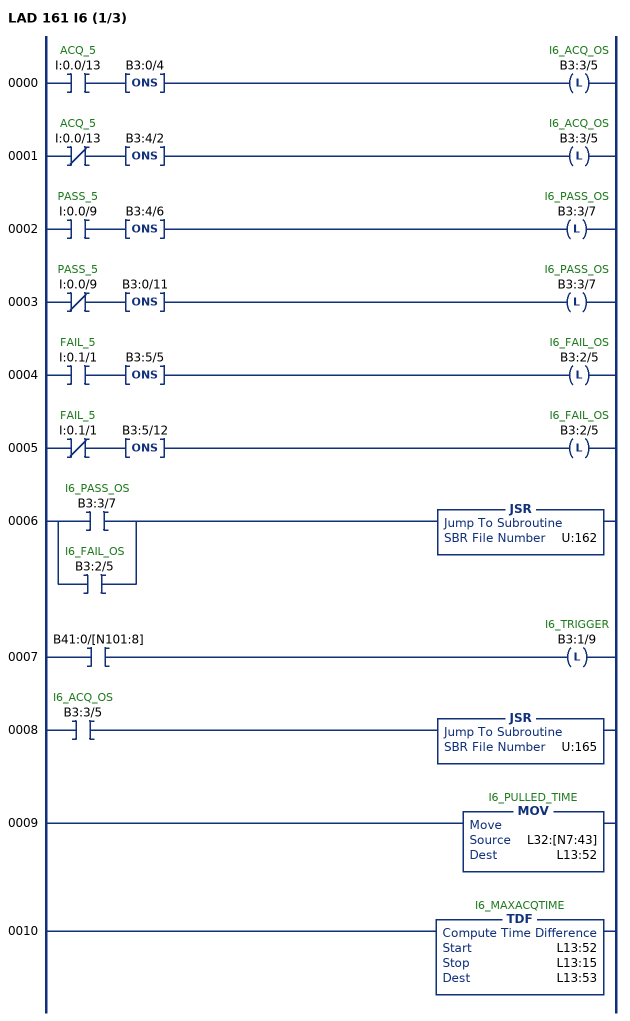
% Rung: 0 %
SOR XIC I:0.0/13 ONS B3:0/4 OTL B3:3/5 EOR
%   I:0.0/13  ACQ_5 %
%   B3:3/5  I6_ACQ_OS %
% Rung: 1 %
SOR XIO I:0.0/13 ONS B3:4/2 OTL B3:3/5 EOR
%   I:0.0/13  ACQ_5 %
%   B3:3/5  I6_ACQ_OS %
% Rung: 2 %
SOR XIC I:0.0/9 ONS B3:4/6 OTL B3:3/7 EOR
%   I:0.0/9  PASS_5 %
%   B3:3/7  I6_PASS_OS %
% Rung: 3 %
SOR XIO I:0.0/9 ONS B3:0/11 OTL B3:3/7 EOR
%   I:0.0/9  PASS_5 %
%   B3:3/7  I6_PASS_OS %
% Rung: 4 %
SOR XIC I:0.1/1 ONS B3:5/5 OTL B3:2/5 EOR
%   I:0.1/1  FAIL_5 %
%   B3:2/5  I6_FAIL_OS %
% Rung: 5 %
SOR XIO I:0.1/1 ONS B3:5/12 OTL B3:2/5 EOR
%   I:0.1/1  FAIL_5 %
%   B3:2/5  I6_FAIL_OS %
% Rung: 6 %
SOR BST XIC B3:3/7 NXB XIC B3:2/5 BND JSR U:162 EOR
%   B3:3/7  I6_PASS_OS %
%   B3:2/5  I6_FAIL_OS %
% Rung: 7 %
SOR XIC B41:0/[N101:8] OTL B3:1/9 EOR
%   B41:0  TOP_OK_3 %
%   N101:8  I6_TRIG_LOC %
%   B3:1/9  I6_TRIGGER %
% Rung: 8 %
SOR XIC B3:3/5 JSR U:165 EOR
%   B3:3/5  I6_ACQ_OS %
% Rung: 9 %
SOR MOV L32:[N7:43] L13:52 EOR
%   N7:43  I6_OLDEST_PART_INDEX %
%   L13:52  I6_PULLED_TIME %
% Rung: 10 %
SOR TDF L13:52 L13:15 L13:53 EOR
%   L13:52  I6_PULLED_TIME %
%   L13:15  THE_TIME %
%   L13:53  I6_MAXACQTIME %

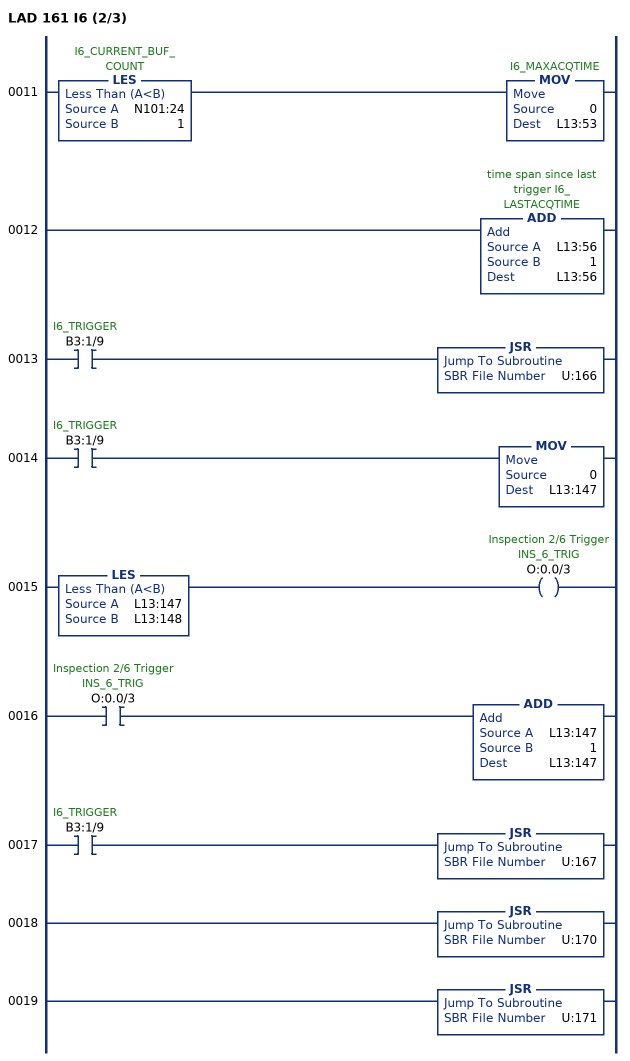
% Rung: 11 %
SOR LES N101:24 1 MOV 0 L13:53 EOR
%   N101:24  I6_CURRENT_BUF_COUNT %
%   L13:53  I6_MAXACQTIME %
% Rung: 12 %
SOR ADD L13:56 1 L13:56 EOR
%   L13:56  I6_LASTACQTIME  "time span since last trigger" %
% Rung: 13 %
SOR XIC B3:1/9 JSR U:166 EOR
%   B3:1/9  I6_TRIGGER %
% Rung: 14 %
SOR XIC B3:1/9 MOV 0 L13:147 EOR
%   B3:1/9  I6_TRIGGER %
% Rung: 15 %
SOR LES L13:147 L13:148 OTE O:0.0/3 EOR
%   O:0.0/3  INS_6_TRIG  "Inspection 2/6 Trigger" %
% Rung: 16 %
SOR XIC O:0.0/3 ADD L13:147 1 L13:147 EOR
%   O:0.0/3  INS_6_TRIG  "Inspection 2/6 Trigger" %
% Rung: 17 %
SOR XIC B3:1/9 JSR U:167 EOR
%   B3:1/9  I6_TRIGGER %
% Rung: 18 %
SOR JSR U:170 EOR
% Rung: 19 %
SOR JSR U:171 EOR

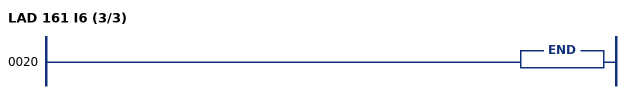
% Rung: 20 %
SOR END EOR

LADDER 162 "I6 RESULT"
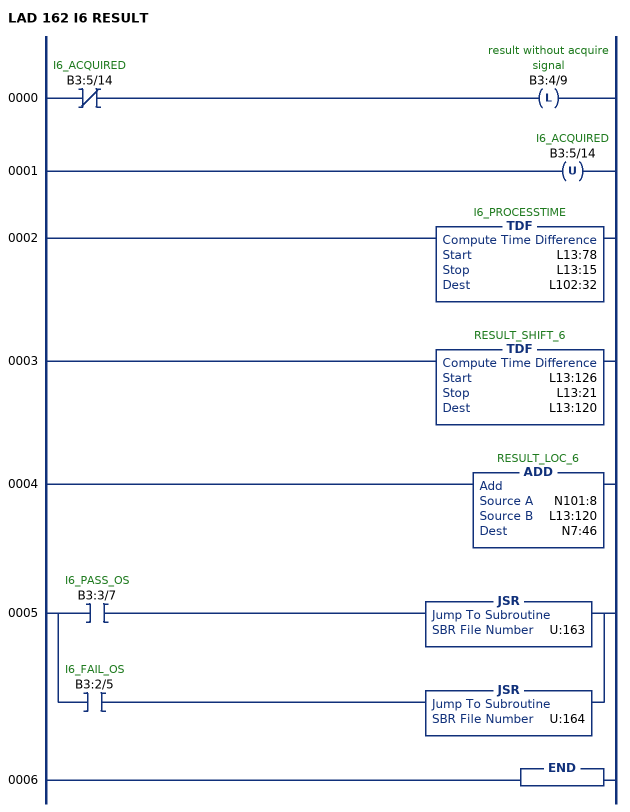
% Rung: 0 %
SOR XIO B3:5/14 OTL B3:4/9 EOR
%   B3:5/14  I6_ACQUIRED %
%   B3:4/9  "result without acquire signal" %
% Rung: 1 %
SOR OTU B3:5/14 EOR
%   B3:5/14  I6_ACQUIRED %
% Rung: 2 %
SOR TDF L13:78 L13:15 L102:32 EOR
%   L13:78  I6_TIMEOFACQ %
%   L13:15  THE_TIME %
%   L102:32  I6_PROCESSTIME %
% Rung: 3 %
SOR TDF L13:126 L13:21 L13:120 EOR
%   L13:126  I6_PROCESS_START_POS %
%   L13:21  TOP_POSITION %
%   L13:120  RESULT_SHIFT_6 %
% Rung: 4 %
SOR ADD N101:8 L13:120 N7:46 EOR
%   N101:8  I6_TRIG_LOC %
%   L13:120  RESULT_SHIFT_6 %
%   N7:46  RESULT_LOC_6 %
% Rung: 5 %
SOR BST XIC B3:3/7 JSR U:163 NXB XIC B3:2/5 JSR U:164 BND EOR
%   B3:3/7  I6_PASS_OS %
%   B3:2/5  I6_FAIL_OS %
% Rung: 6 %
SOR END EOR

LADDER 163 "I6 PASS"
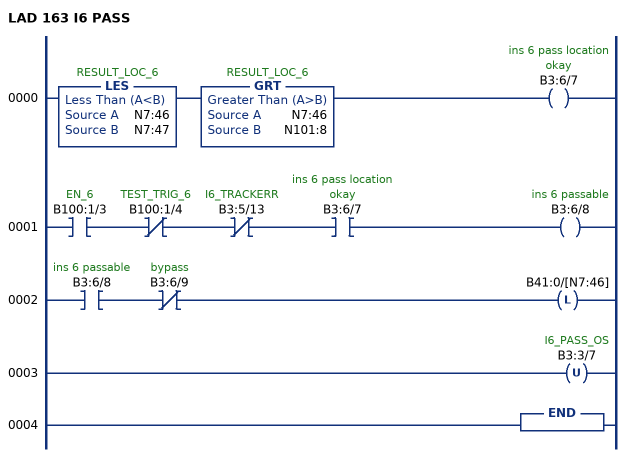
% Rung: 0 %
SOR LES N7:46 N7:47 GRT N7:46 N101:8 OTE B3:6/7 EOR
%   N7:46  RESULT_LOC_6 %
%   N7:47  I6_MAX_SHIFT  "ins 6 maximum result location" %
%   N101:8  I6_TRIG_LOC %
%   B3:6/7  "ins 6 pass location okay" %
% Rung: 1 %
SOR XIC B100:1/3 XIO B100:1/4 XIO B3:5/13 XIC B3:6/7 OTE B3:6/8 EOR
%   B100:1/3  EN_6 %
%   B100:1/4  TEST_TRIG_6 %
%   B3:5/13  I6_TRACKERR %
%   B3:6/7  "ins 6 pass location okay" %
%   B3:6/8  "ins 6 passable" %
% Rung: 2 %
SOR XIC B3:6/8 XIO B3:6/9 OTL B41:0/[N7:46] EOR
%   B3:6/8  "ins 6 passable" %
%   B3:6/9  "bypass" %
%   B41:0  TOP_OK_3 %
%   N7:46  RESULT_LOC_6 %
% Rung: 3 %
SOR OTU B3:3/7 EOR
%   B3:3/7  I6_PASS_OS %
% Rung: 4 %
SOR END EOR

LADDER 164 "I6 FAIL"
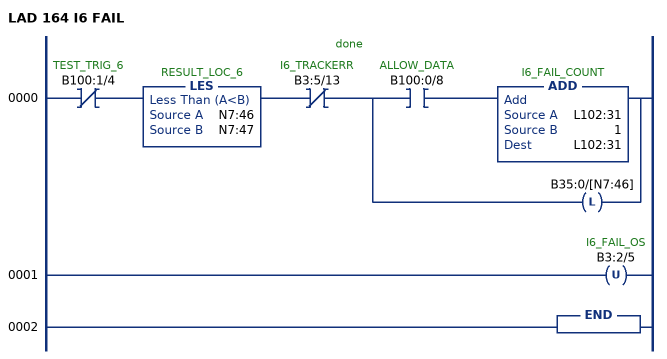
% Rung: 0 %
% done %
SOR XIO B100:1/4 LES N7:46 N7:47 XIO B3:5/13 BST XIC B100:0/8 ADD L102:31 1 L102:31 NXB OTL B35:0/[N7:46] BND EOR
%   B100:1/4  TEST_TRIG_6 %
%   N7:46  RESULT_LOC_6 %
%   N7:47  I6_MAX_SHIFT  "ins 6 maximum result location" %
%   B3:5/13  I6_TRACKERR %
%   B100:0/8  ALLOW_DATA %
%   L102:31  I6_FAIL_COUNT %
%   B35:0  TOP_NG %
% Rung: 1 %
SOR OTU B3:2/5 EOR
%   B3:2/5  I6_FAIL_OS %
% Rung: 2 %
SOR END EOR

LADDER 165 "I6 ACQ"
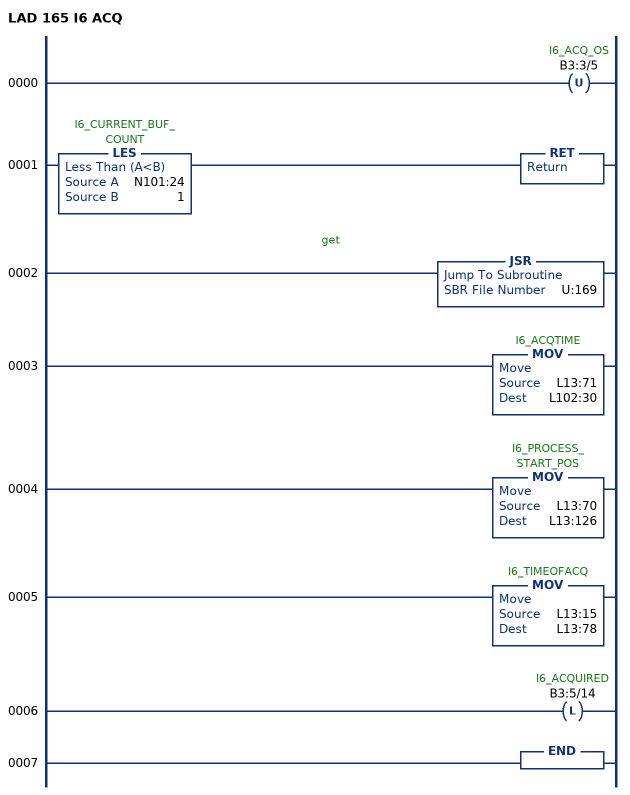
% Rung: 0 %
SOR OTU B3:3/5 EOR
%   B3:3/5  I6_ACQ_OS %
% Rung: 1 %
SOR LES N101:24 1 RET EOR
%   N101:24  I6_CURRENT_BUF_COUNT %
% Rung: 2 %
% get %
SOR JSR U:169 EOR
% Rung: 3 %
SOR MOV L13:71 L102:30 EOR
%   L13:71  I6_TIME_SPAN %
%   L102:30  I6_ACQTIME %
% Rung: 4 %
SOR MOV L13:70 L13:126 EOR
%   L13:70  I6_PULLED_POSITION %
%   L13:126  I6_PROCESS_START_POS %
% Rung: 5 %
SOR MOV L13:15 L13:78 EOR
%   L13:15  THE_TIME %
%   L13:78  I6_TIMEOFACQ %
% Rung: 6 %
SOR OTL B3:5/14 EOR
%   B3:5/14  I6_ACQUIRED %
% Rung: 7 %
SOR END EOR

LADDER 166 "I6 TESTER"
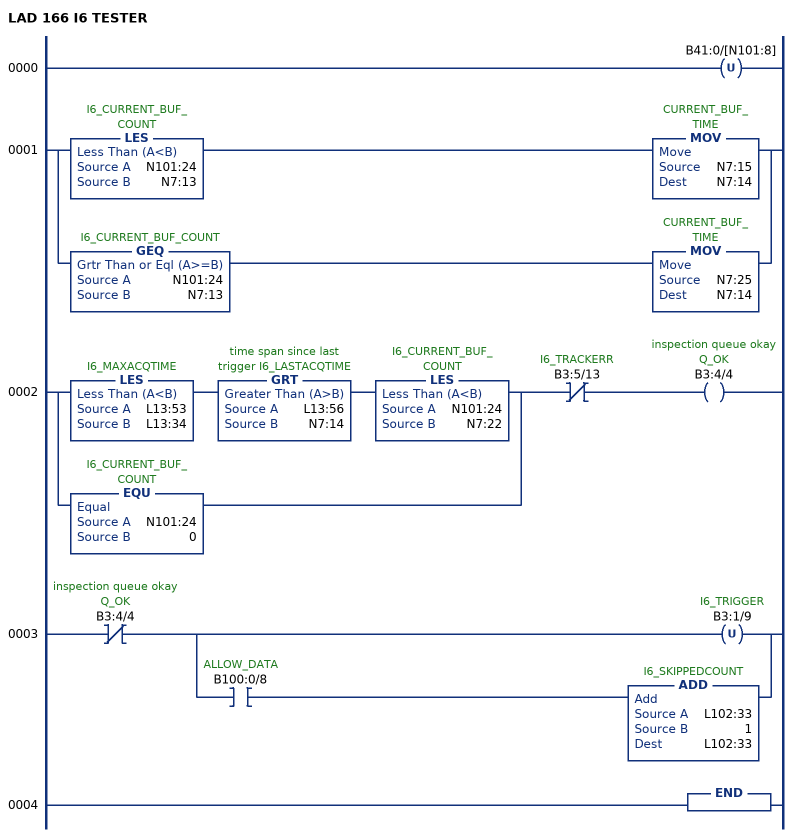
% Rung: 0 %
SOR OTU B41:0/[N101:8] EOR
%   B41:0  TOP_OK_3 %
%   N101:8  I6_TRIG_LOC %
% Rung: 1 %
SOR BST LES N101:24 N7:13 MOV N7:15 N7:14 NXB GEQ N101:24 N7:13 MOV N7:25 N7:14 BND EOR
%   N101:24  I6_CURRENT_BUF_COUNT %
%   N7:13  BUF_TRANS  "cam to pc buf transition" %
%   N7:15  CAM_BUF_TIME  "cam buf time" %
%   N7:14  CURRENT_BUF_TIME %
%   N7:25  PC_BUF_TIME  "pc buf time" %
% Rung: 2 %
SOR BST LES L13:53 L13:34 GRT L13:56 N7:14 LES N101:24 N7:22 NXB EQU N101:24 0 BND XIO B3:5/13 OTE B3:4/4 EOR
%   L13:53  I6_MAXACQTIME %
%   L13:34  MAX_ACQ_ALL  "absolute max acquire time before bypass trigger" %
%   L13:56  I6_LASTACQTIME  "time span since last trigger" %
%   N7:14  CURRENT_BUF_TIME %
%   N101:24  I6_CURRENT_BUF_COUNT %
%   N7:22  MAX_BUF_ALL  "max buffer count alowed before bypass" %
%   B3:5/13  I6_TRACKERR %
%   B3:4/4  Q_OK  "inspection queue okay" %
% Rung: 3 %
SOR XIO B3:4/4 BST OTU B3:1/9 NXB XIC B100:0/8 ADD L102:33 1 L102:33 BND EOR
%   B3:4/4  Q_OK  "inspection queue okay" %
%   B3:1/9  I6_TRIGGER %
%   B100:0/8  ALLOW_DATA %
%   L102:33  I6_SKIPPEDCOUNT %
% Rung: 4 %
SOR END EOR

LADDER 167 "I6 TRIG"
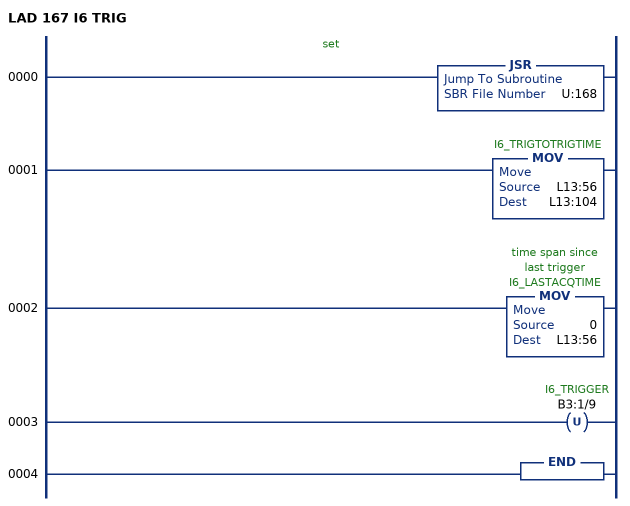
% Rung: 0 %
% set %
SOR JSR U:168 EOR
% Rung: 1 %
SOR MOV L13:56 L13:104 EOR
%   L13:56  I6_LASTACQTIME  "time span since last trigger" %
%   L13:104  I6_TRIGTOTRIGTIME %
% Rung: 2 %
SOR MOV 0 L13:56 EOR
%   L13:56  I6_LASTACQTIME  "time span since last trigger" %
% Rung: 3 %
SOR OTU B3:1/9 EOR
%   B3:1/9  I6_TRIGGER %
% Rung: 4 %
SOR END EOR

LADDER 168 "I6 FIFOSET"
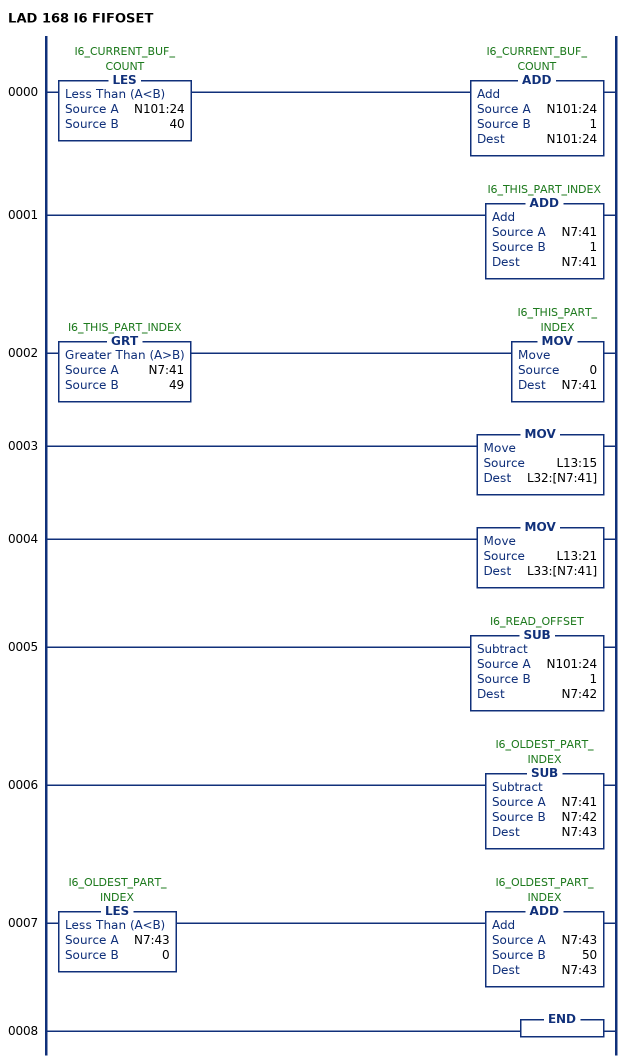
% Rung: 0 %
SOR LES N101:24 40 ADD N101:24 1 N101:24 EOR
%   N101:24  I6_CURRENT_BUF_COUNT %
% Rung: 1 %
SOR ADD N7:41 1 N7:41 EOR
%   N7:41  I6_THIS_PART_INDEX %
% Rung: 2 %
SOR GRT N7:41 49 MOV 0 N7:41 EOR
%   N7:41  I6_THIS_PART_INDEX %
% Rung: 3 %
SOR MOV L13:15 L32:[N7:41] EOR
%   L13:15  THE_TIME %
%   N7:41  I6_THIS_PART_INDEX %
% Rung: 4 %
SOR MOV L13:21 L33:[N7:41] EOR
%   L13:21  TOP_POSITION %
%   N7:41  I6_THIS_PART_INDEX %
% Rung: 5 %
SOR SUB N101:24 1 N7:42 EOR
%   N101:24  I6_CURRENT_BUF_COUNT %
%   N7:42  I6_READ_OFFSET %
% Rung: 6 %
SOR SUB N7:41 N7:42 N7:43 EOR
%   N7:41  I6_THIS_PART_INDEX %
%   N7:42  I6_READ_OFFSET %
%   N7:43  I6_OLDEST_PART_INDEX %
% Rung: 7 %
SOR LES N7:43 0 ADD N7:43 50 N7:43 EOR
%   N7:43  I6_OLDEST_PART_INDEX %
% Rung: 8 %
SOR END EOR

LADDER 169 "I6 FIFOGET"
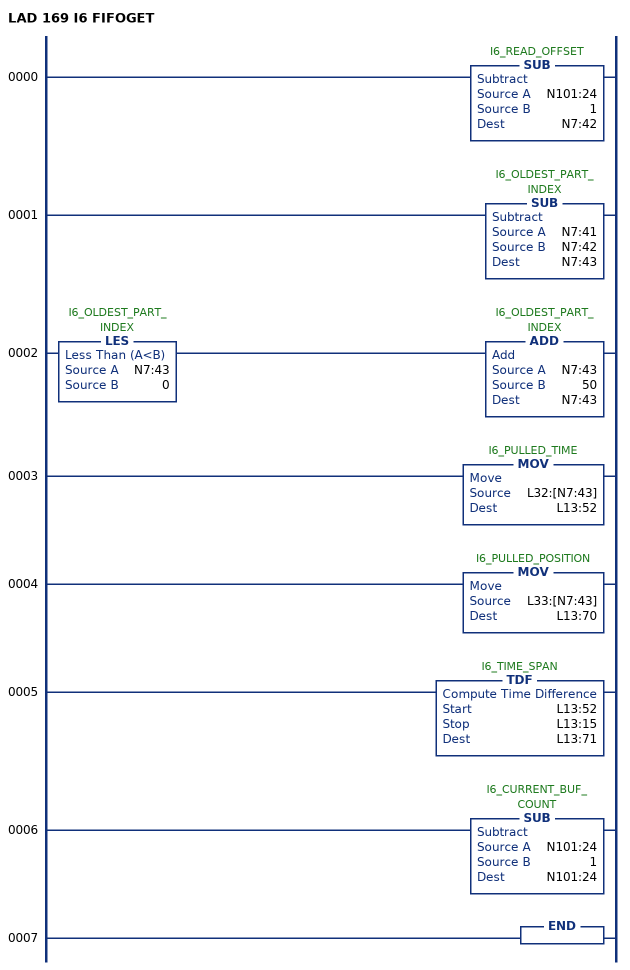
% Rung: 0 %
SOR SUB N101:24 1 N7:42 EOR
%   N101:24  I6_CURRENT_BUF_COUNT %
%   N7:42  I6_READ_OFFSET %
% Rung: 1 %
SOR SUB N7:41 N7:42 N7:43 EOR
%   N7:41  I6_THIS_PART_INDEX %
%   N7:42  I6_READ_OFFSET %
%   N7:43  I6_OLDEST_PART_INDEX %
% Rung: 2 %
SOR LES N7:43 0 ADD N7:43 50 N7:43 EOR
%   N7:43  I6_OLDEST_PART_INDEX %
% Rung: 3 %
SOR MOV L32:[N7:43] L13:52 EOR
%   N7:43  I6_OLDEST_PART_INDEX %
%   L13:52  I6_PULLED_TIME %
% Rung: 4 %
SOR MOV L33:[N7:43] L13:70 EOR
%   N7:43  I6_OLDEST_PART_INDEX %
%   L13:70  I6_PULLED_POSITION %
% Rung: 5 %
SOR TDF L13:52 L13:15 L13:71 EOR
%   L13:52  I6_PULLED_TIME %
%   L13:15  THE_TIME %
%   L13:71  I6_TIME_SPAN %
% Rung: 6 %
SOR SUB N101:24 1 N101:24 EOR
%   N101:24  I6_CURRENT_BUF_COUNT %
% Rung: 7 %
SOR END EOR

LADDER 170 "I6 DATA"
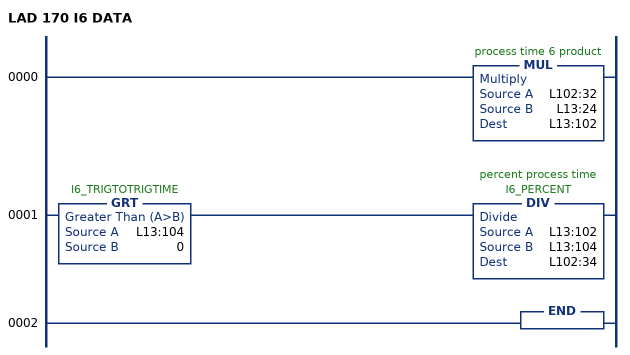
% Rung: 0 %
SOR MUL L102:32 L13:24 L13:102 EOR
%   L102:32  I6_PROCESSTIME %
%   L13:24  "multiplyer to make devision come out to a percentage" %
%   L13:102  "process time 6 product" %
% Rung: 1 %
SOR GRT L13:104 0 DIV L13:102 L13:104 L102:34 EOR
%   L13:104  I6_TRIGTOTRIGTIME %
%   L13:102  "process time 6 product" %
%   L102:34  I6_PERCENT  "percent process time" %
% Rung: 2 %
SOR END EOR

LADDER 171 "I6 FAULT"
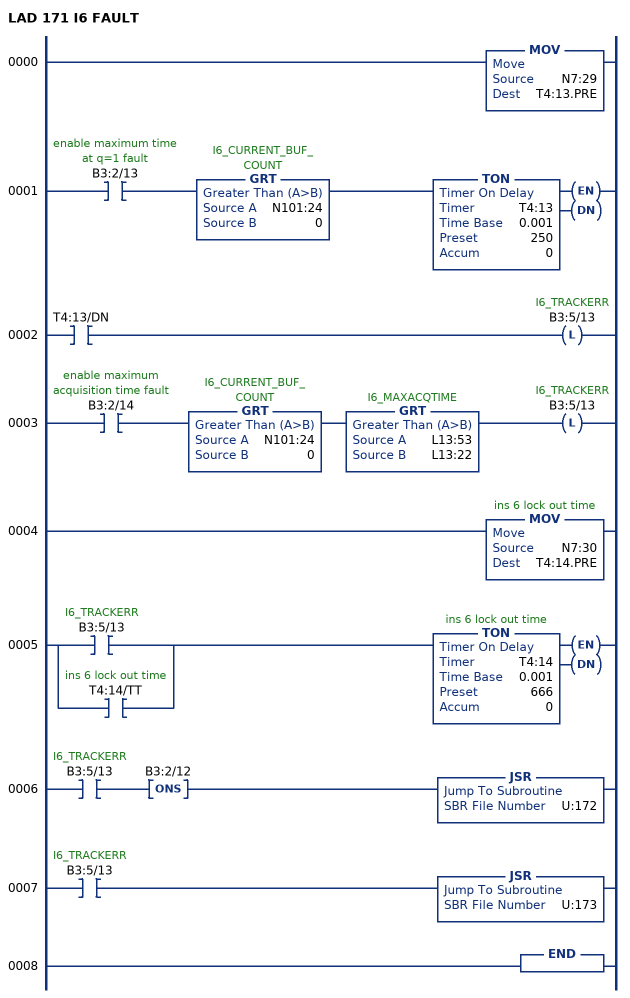
% Rung: 0 %
SOR MOV N7:29 T4:13.PRE EOR
%   N7:29  "max allowed ms time for q to be above 1 if safe fault is used" %
% Rung: 1 %
SOR XIC B3:2/13 GRT N101:24 0 TON T4:13 0.001 250 0 EOR
%   B3:2/13  "enable maximum time at q=1 fault" %
%   N101:24  I6_CURRENT_BUF_COUNT %
% Rung: 2 %
SOR XIC T4:13/DN OTL B3:5/13 EOR
%   B3:5/13  I6_TRACKERR %
% Rung: 3 %
SOR XIC B3:2/14 GRT N101:24 0 GRT L13:53 L13:22 OTL B3:5/13 EOR
%   B3:2/14  "enable maximum acquisition time fault" %
%   N101:24  I6_CURRENT_BUF_COUNT %
%   L13:53  I6_MAXACQTIME %
%   L13:22  "maximum of the longest acquire time allowed if maximum acquire time fault is enabled" %
%   B3:5/13  I6_TRACKERR %
% Rung: 4 %
SOR MOV N7:30 T4:14.PRE EOR
%   N7:30  "ms time setting to lock out inspection to give all pending images a chance to clear" %
%   T4:14  "ins 6 lock out time" %
% Rung: 5 %
SOR BST XIC B3:5/13 NXB XIC T4:14/TT BND TON T4:14 0.001 666 0 EOR
%   B3:5/13  I6_TRACKERR %
%   T4:14  "ins 6 lock out time" %
% Rung: 6 %
SOR XIC B3:5/13 ONS B3:2/12 JSR U:172 EOR
%   B3:5/13  I6_TRACKERR %
% Rung: 7 %
SOR XIC B3:5/13 JSR U:173 EOR
%   B3:5/13  I6_TRACKERR %
% Rung: 8 %
SOR END EOR

LADDER 172 "I6 FIX1"
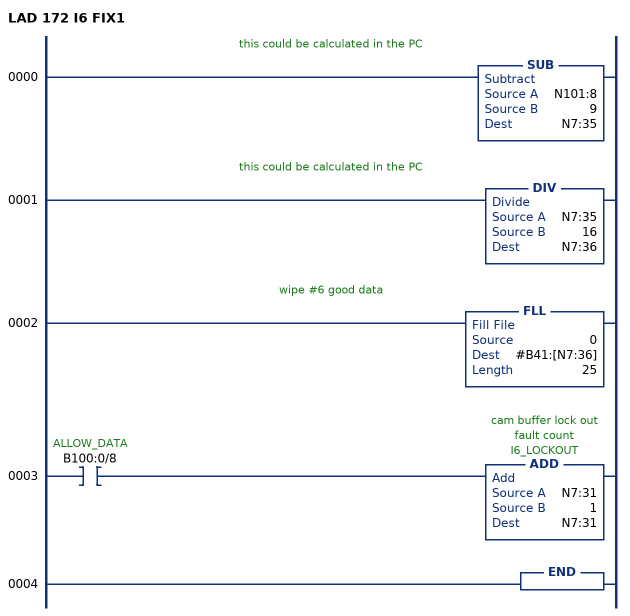
% Rung: 0 %
% this could be calculated in the PC %
SOR SUB N101:8 9 N7:35 EOR
%   N101:8  I6_TRIG_LOC %
% Rung: 1 %
% this could be calculated in the PC %
SOR DIV N7:35 16 N7:36 EOR
% Rung: 2 %
% wipe #6 good data %
SOR FLL 0 #B41:[N7:36] 25 EOR
% Rung: 3 %
SOR XIC B100:0/8 ADD N7:31 1 N7:31 EOR
%   B100:0/8  ALLOW_DATA %
%   N7:31  I6_LOCKOUT  "cam buffer lock out fault count" %
% Rung: 4 %
SOR END EOR

LADDER 173 "I6 FIX2"
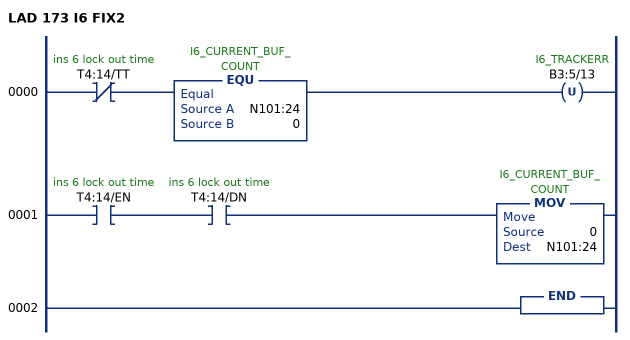
% Rung: 0 %
SOR XIO T4:14/TT EQU N101:24 0 OTU B3:5/13 EOR
%   T4:14  "ins 6 lock out time" %
%   N101:24  I6_CURRENT_BUF_COUNT %
%   B3:5/13  I6_TRACKERR %
% Rung: 1 %
SOR XIC T4:14/EN XIC T4:14/DN MOV 0 N101:24 EOR
%   T4:14  "ins 6 lock out time" %
%   N101:24  I6_CURRENT_BUF_COUNT %
% Rung: 2 %
SOR END EOR

LADDER 174 "I7"
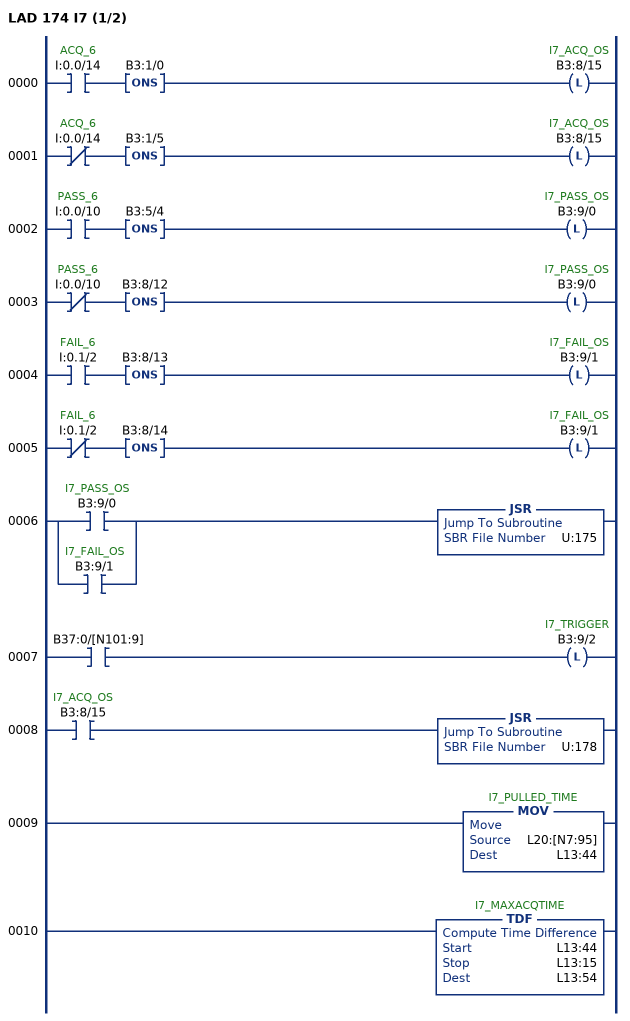
% Rung: 0 %
SOR XIC I:0.0/14 ONS B3:1/0 OTL B3:8/15 EOR
%   I:0.0/14  ACQ_6 %
%   B3:8/15  I7_ACQ_OS %
% Rung: 1 %
SOR XIO I:0.0/14 ONS B3:1/5 OTL B3:8/15 EOR
%   I:0.0/14  ACQ_6 %
%   B3:8/15  I7_ACQ_OS %
% Rung: 2 %
SOR XIC I:0.0/10 ONS B3:5/4 OTL B3:9/0 EOR
%   I:0.0/10  PASS_6 %
%   B3:9/0  I7_PASS_OS %
% Rung: 3 %
SOR XIO I:0.0/10 ONS B3:8/12 OTL B3:9/0 EOR
%   I:0.0/10  PASS_6 %
%   B3:9/0  I7_PASS_OS %
% Rung: 4 %
SOR XIC I:0.1/2 ONS B3:8/13 OTL B3:9/1 EOR
%   I:0.1/2  FAIL_6 %
%   B3:9/1  I7_FAIL_OS %
% Rung: 5 %
SOR XIO I:0.1/2 ONS B3:8/14 OTL B3:9/1 EOR
%   I:0.1/2  FAIL_6 %
%   B3:9/1  I7_FAIL_OS %
% Rung: 6 %
SOR BST XIC B3:9/0 NXB XIC B3:9/1 BND JSR U:175 EOR
%   B3:9/0  I7_PASS_OS %
%   B3:9/1  I7_FAIL_OS %
% Rung: 7 %
SOR XIC B37:0/[N101:9] OTL B3:9/2 EOR
%   B37:0  TOP_OK_1 %
%   N101:9  I7_TRIG_LOC %
%   B3:9/2  I7_TRIGGER %
% Rung: 8 %
SOR XIC B3:8/15 JSR U:178 EOR
%   B3:8/15  I7_ACQ_OS %
% Rung: 9 %
SOR MOV L20:[N7:95] L13:44 EOR
%   N7:95  I7_OLDEST_PART_INDEX %
%   L13:44  I7_PULLED_TIME %
% Rung: 10 %
SOR TDF L13:44 L13:15 L13:54 EOR
%   L13:44  I7_PULLED_TIME %
%   L13:15  THE_TIME %
%   L13:54  I7_MAXACQTIME %

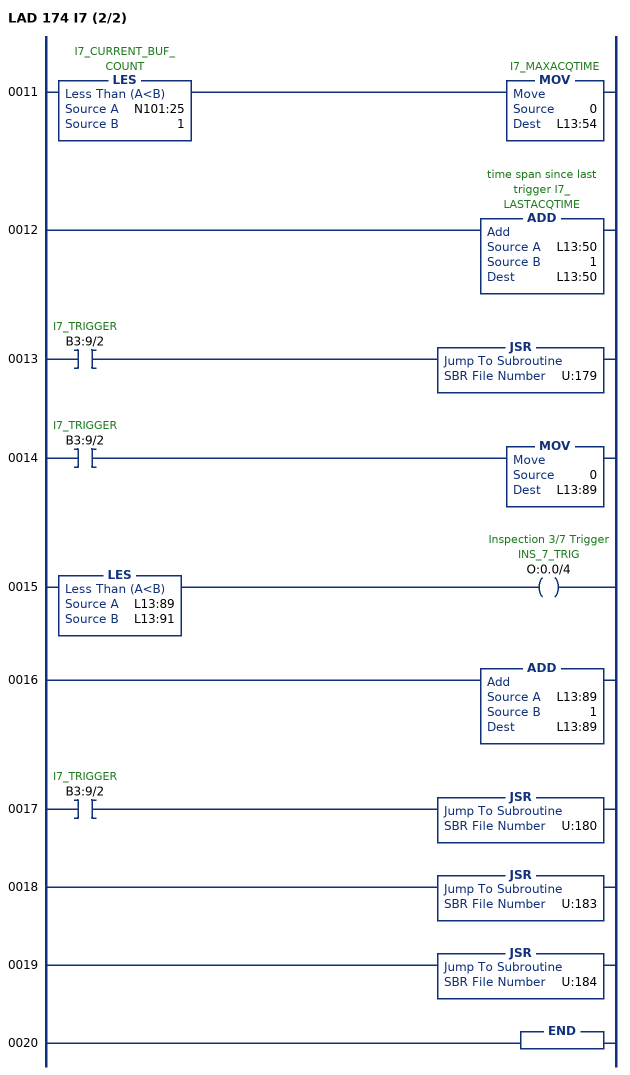
% Rung: 11 %
SOR LES N101:25 1 MOV 0 L13:54 EOR
%   N101:25  I7_CURRENT_BUF_COUNT %
%   L13:54  I7_MAXACQTIME %
% Rung: 12 %
SOR ADD L13:50 1 L13:50 EOR
%   L13:50  I7_LASTACQTIME  "time span since last trigger" %
% Rung: 13 %
SOR XIC B3:9/2 JSR U:179 EOR
%   B3:9/2  I7_TRIGGER %
% Rung: 14 %
SOR XIC B3:9/2 MOV 0 L13:89 EOR
%   B3:9/2  I7_TRIGGER %
% Rung: 15 %
SOR LES L13:89 L13:91 OTE O:0.0/4 EOR
%   L13:91  "test fire interval index" %
%   O:0.0/4  INS_7_TRIG  "Inspection 3/7 Trigger" %
% Rung: 16 %
SOR ADD L13:89 1 L13:89 EOR
% Rung: 17 %
SOR XIC B3:9/2 JSR U:180 EOR
%   B3:9/2  I7_TRIGGER %
% Rung: 18 %
SOR JSR U:183 EOR
% Rung: 19 %
SOR JSR U:184 EOR
% Rung: 20 %
SOR END EOR

LADDER 175 "I7 RESULT"
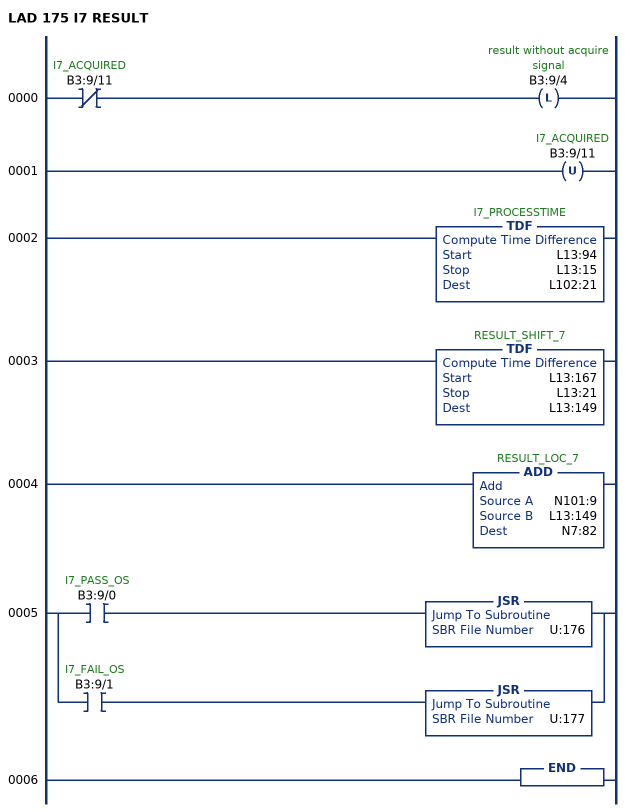
% Rung: 0 %
SOR XIO B3:9/11 OTL B3:9/4 EOR
%   B3:9/11  I7_ACQUIRED %
%   B3:9/4  "result without acquire signal" %
% Rung: 1 %
SOR OTU B3:9/11 EOR
%   B3:9/11  I7_ACQUIRED %
% Rung: 2 %
SOR TDF L13:94 L13:15 L102:21 EOR
%   L13:94  I7_TIMEOFACQ %
%   L13:15  THE_TIME %
%   L102:21  I7_PROCESSTIME %
% Rung: 3 %
SOR TDF L13:167 L13:21 L13:149 EOR
%   L13:167  I7_PROCESS_START_POS %
%   L13:21  TOP_POSITION %
%   L13:149  RESULT_SHIFT_7 %
% Rung: 4 %
SOR ADD N101:9 L13:149 N7:82 EOR
%   N101:9  I7_TRIG_LOC %
%   L13:149  RESULT_SHIFT_7 %
%   N7:82  RESULT_LOC_7 %
% Rung: 5 %
SOR BST XIC B3:9/0 JSR U:176 NXB XIC B3:9/1 JSR U:177 BND EOR
%   B3:9/0  I7_PASS_OS %
%   B3:9/1  I7_FAIL_OS %
% Rung: 6 %
SOR END EOR

LADDER 176 "I7 PASS"
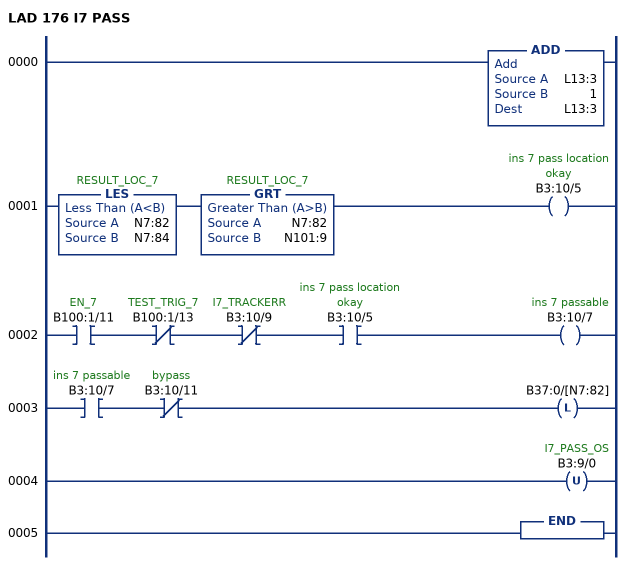
% Rung: 0 %
SOR ADD L13:3 1 L13:3 EOR
% Rung: 1 %
SOR LES N7:82 N7:84 GRT N7:82 N101:9 OTE B3:10/5 EOR
%   N7:82  RESULT_LOC_7 %
%   N7:84  I7_MAX_SHIFT %
%   N101:9  I7_TRIG_LOC %
%   B3:10/5  "ins 7 pass location okay" %
% Rung: 2 %
SOR XIC B100:1/11 XIO B100:1/13 XIO B3:10/9 XIC B3:10/5 OTE B3:10/7 EOR
%   B100:1/11  EN_7 %
%   B100:1/13  TEST_TRIG_7 %
%   B3:10/9  I7_TRACKERR %
%   B3:10/5  "ins 7 pass location okay" %
%   B3:10/7  "ins 7 passable" %
% Rung: 3 %
SOR XIC B3:10/7 XIO B3:10/11 OTL B37:0/[N7:82] EOR
%   B3:10/7  "ins 7 passable" %
%   B3:10/11  "bypass" %
%   B37:0  TOP_OK_1 %
%   N7:82  RESULT_LOC_7 %
% Rung: 4 %
SOR OTU B3:9/0 EOR
%   B3:9/0  I7_PASS_OS %
% Rung: 5 %
SOR END EOR

LADDER 177 "I7 FAIL"
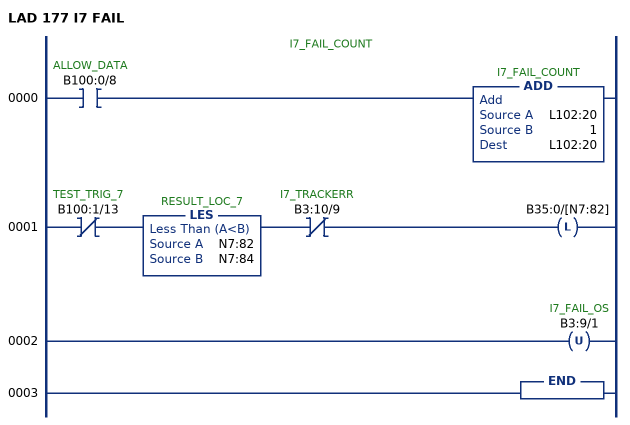
% Rung: 0 %
% I7_FAIL_COUNT %
SOR XIC B100:0/8 ADD L102:20 1 L102:20 EOR
%   B100:0/8  ALLOW_DATA %
%   L102:20  I7_FAIL_COUNT %
% Rung: 1 %
SOR XIO B100:1/13 LES N7:82 N7:84 XIO B3:10/9 OTL B35:0/[N7:82] EOR
%   B100:1/13  TEST_TRIG_7 %
%   N7:82  RESULT_LOC_7 %
%   N7:84  I7_MAX_SHIFT %
%   B3:10/9  I7_TRACKERR %
%   B35:0  TOP_NG %
% Rung: 2 %
SOR OTU B3:9/1 EOR
%   B3:9/1  I7_FAIL_OS %
% Rung: 3 %
SOR END EOR

LADDER 178 "I7 ACQ"
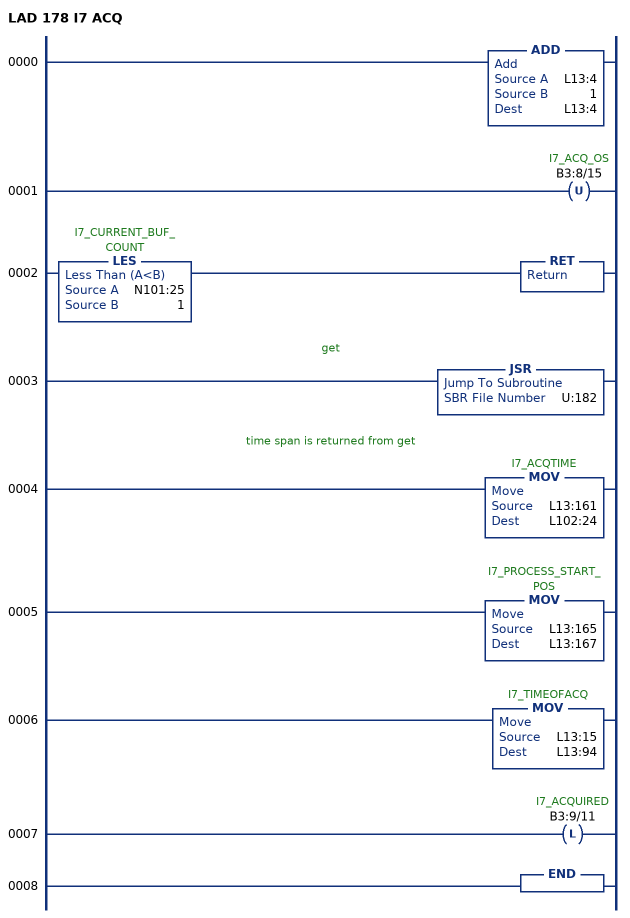
% Rung: 0 %
SOR ADD L13:4 1 L13:4 EOR
% Rung: 1 %
SOR OTU B3:8/15 EOR
%   B3:8/15  I7_ACQ_OS %
% Rung: 2 %
SOR LES N101:25 1 RET EOR
%   N101:25  I7_CURRENT_BUF_COUNT %
% Rung: 3 %
% get %
SOR JSR U:182 EOR
% Rung: 4 %
% time span is returned from get %
SOR MOV L13:161 L102:24 EOR
%   L13:161  I7_TIME_SPAN %
%   L102:24  I7_ACQTIME %
% Rung: 5 %
SOR MOV L13:165 L13:167 EOR
%   L13:165  I7_PULLED_POSITION %
%   L13:167  I7_PROCESS_START_POS %
% Rung: 6 %
SOR MOV L13:15 L13:94 EOR
%   L13:15  THE_TIME %
%   L13:94  I7_TIMEOFACQ %
% Rung: 7 %
SOR OTL B3:9/11 EOR
%   B3:9/11  I7_ACQUIRED %
% Rung: 8 %
SOR END EOR

LADDER 179 "I7 TESTER"
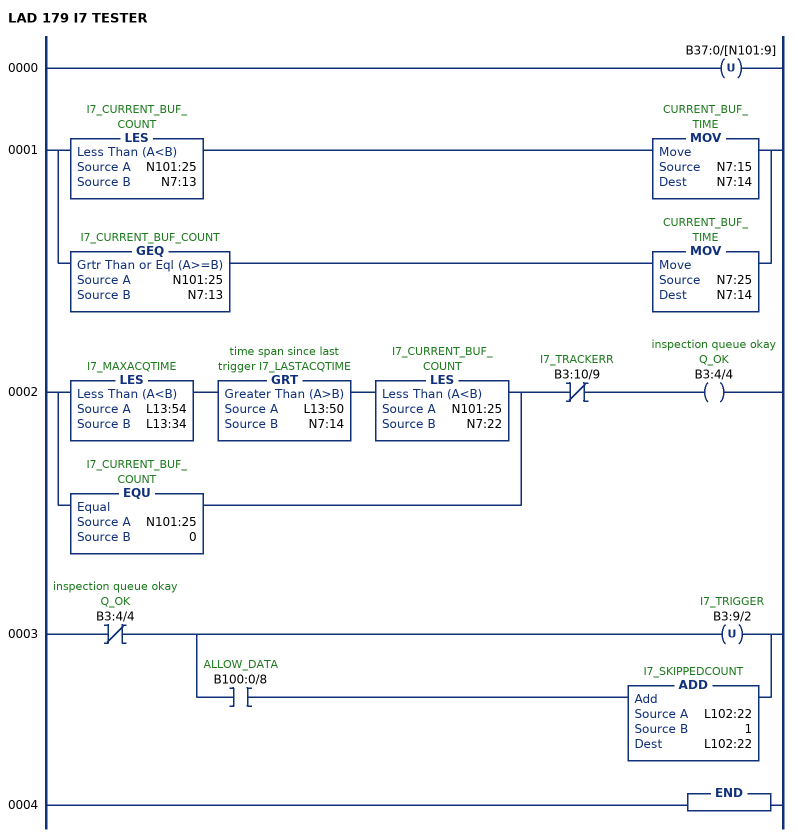
% Rung: 0 %
SOR OTU B37:0/[N101:9] EOR
%   B37:0  TOP_OK_1 %
%   N101:9  I7_TRIG_LOC %
% Rung: 1 %
SOR BST LES N101:25 N7:13 MOV N7:15 N7:14 NXB GEQ N101:25 N7:13 MOV N7:25 N7:14 BND EOR
%   N101:25  I7_CURRENT_BUF_COUNT %
%   N7:13  BUF_TRANS  "cam to pc buf transition" %
%   N7:15  CAM_BUF_TIME  "cam buf time" %
%   N7:14  CURRENT_BUF_TIME %
%   N7:25  PC_BUF_TIME  "pc buf time" %
% Rung: 2 %
SOR BST LES L13:54 L13:34 GRT L13:50 N7:14 LES N101:25 N7:22 NXB EQU N101:25 0 BND XIO B3:10/9 OTE B3:4/4 EOR
%   L13:54  I7_MAXACQTIME %
%   L13:34  MAX_ACQ_ALL  "absolute max acquire time before bypass trigger" %
%   L13:50  I7_LASTACQTIME  "time span since last trigger" %
%   N7:14  CURRENT_BUF_TIME %
%   N101:25  I7_CURRENT_BUF_COUNT %
%   N7:22  MAX_BUF_ALL  "max buffer count alowed before bypass" %
%   B3:10/9  I7_TRACKERR %
%   B3:4/4  Q_OK  "inspection queue okay" %
% Rung: 3 %
SOR XIO B3:4/4 BST OTU B3:9/2 NXB XIC B100:0/8 ADD L102:22 1 L102:22 BND EOR
%   B3:4/4  Q_OK  "inspection queue okay" %
%   B3:9/2  I7_TRIGGER %
%   B100:0/8  ALLOW_DATA %
%   L102:22  I7_SKIPPEDCOUNT %
% Rung: 4 %
SOR END EOR

LADDER 180 "I7 TRIG"
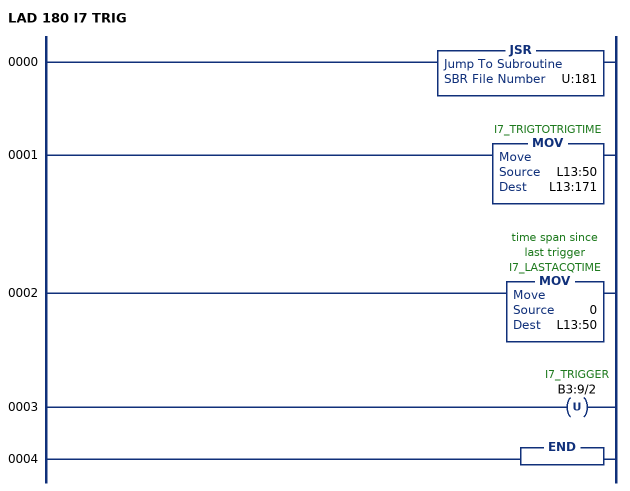
% Rung: 0 %
SOR JSR U:181 EOR
% Rung: 1 %
SOR MOV L13:50 L13:171 EOR
%   L13:50  I7_LASTACQTIME  "time span since last trigger" %
%   L13:171  I7_TRIGTOTRIGTIME %
% Rung: 2 %
SOR MOV 0 L13:50 EOR
%   L13:50  I7_LASTACQTIME  "time span since last trigger" %
% Rung: 3 %
SOR OTU B3:9/2 EOR
%   B3:9/2  I7_TRIGGER %
% Rung: 4 %
SOR END EOR

LADDER 181 "I7 FIFOSET"
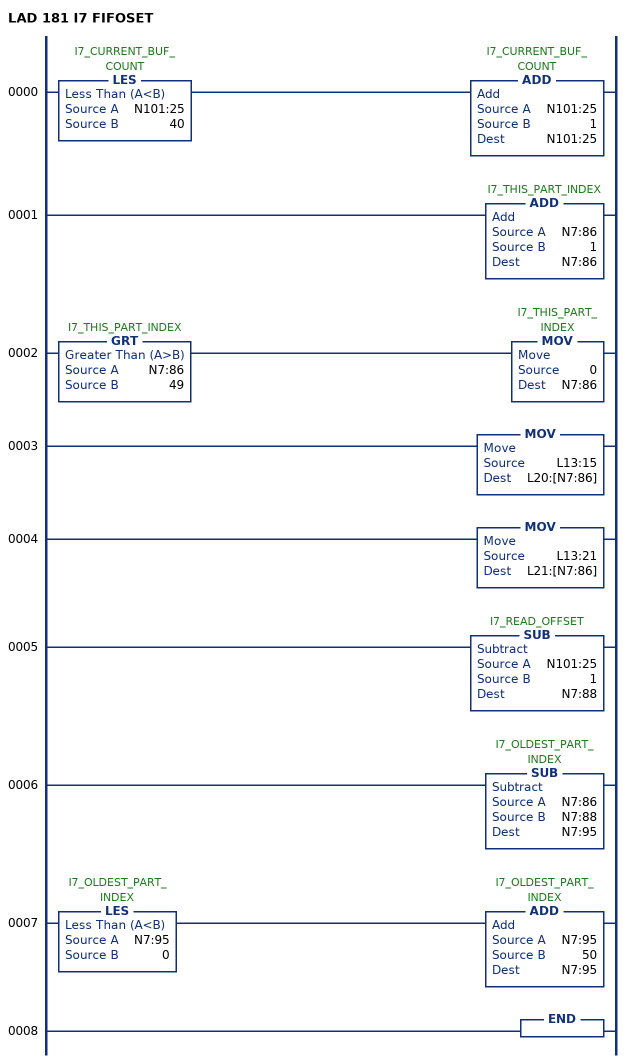
% Rung: 0 %
SOR LES N101:25 40 ADD N101:25 1 N101:25 EOR
%   N101:25  I7_CURRENT_BUF_COUNT %
% Rung: 1 %
SOR ADD N7:86 1 N7:86 EOR
%   N7:86  I7_THIS_PART_INDEX %
% Rung: 2 %
SOR GRT N7:86 49 MOV 0 N7:86 EOR
%   N7:86  I7_THIS_PART_INDEX %
% Rung: 3 %
SOR MOV L13:15 L20:[N7:86] EOR
%   L13:15  THE_TIME %
%   N7:86  I7_THIS_PART_INDEX %
% Rung: 4 %
SOR MOV L13:21 L21:[N7:86] EOR
%   L13:21  TOP_POSITION %
%   N7:86  I7_THIS_PART_INDEX %
% Rung: 5 %
SOR SUB N101:25 1 N7:88 EOR
%   N101:25  I7_CURRENT_BUF_COUNT %
%   N7:88  I7_READ_OFFSET %
% Rung: 6 %
SOR SUB N7:86 N7:88 N7:95 EOR
%   N7:86  I7_THIS_PART_INDEX %
%   N7:88  I7_READ_OFFSET %
%   N7:95  I7_OLDEST_PART_INDEX %
% Rung: 7 %
SOR LES N7:95 0 ADD N7:95 50 N7:95 EOR
%   N7:95  I7_OLDEST_PART_INDEX %
% Rung: 8 %
SOR END EOR

LADDER 182 "I7 FIFOGET"
